// TwinCAT 3 PLC project NCInterpolation
// ProgramVersion: 3.1.0.8
// libraries:
//   Tc2_MC2, * (Beckhoff Automation GmbH)
//   Tc2_NCI, * (Beckhoff Automation GmbH)
//   Tc2_PlcInterpolation, * (Beckhoff Automation GmbH)
//   Tc2_Standard, * (Beckhoff Automation GmbH)
//   Tc2_System, * (Beckhoff Automation GmbH)
//   Tc3_Module, * (Beckhoff Automation GmbH)
// project tree:
//   GVLs/ GVL.TcGVL
//   / PlcTask.TcTTO
//   POUs/ Interpolate.TcPOU, MAIN.TcPOU, P_UML_Grafcet_Sequence.TcPOU
// real-time tasks:
//   TASK PlcTask: cycle T#10ms, priority 20, ADS port 350
// motion (NC):
//   TASK NC-Task 1 SAF: cycle T#5ms, priority 4, ADS port 501
//   TASK NC-Task 1 SVB: cycle T#10ms, priority 9, ADS port 511
//   AXIS FaulHaber_X (id 2)
//     General: UnitName=°
//     Dynamic: Acceleration=1925.33, Deceleration=1925.33, Jerk=187.597, DelayTime=0.015
//     Velo: Maximum=38000
//     OtherSettings: AllowMotionCmdToSlave=true
//     encoder EncType=19
//       EncPara: ScaleFactorNumerator=360, ScaleFactorDenominator=3000, MaxCount=#xffffffff
//         Inc: RefSoftSyncMask=#x0000ffff
//     drive DrvType=16
//       DrvPara: MaxCount=#xffffffff
//         Analog: VeloReferenz=42000
//         TimeComp: TaskDelayCycles=1
//     controller CtrType=1
//       CtrPara: PriorControlFactor=1
//         PosDiffControl: Enable=false
//         Observer: BandWidth=20
//   AXIS Stepper (id 4)
//     General: UnitName=°
//     Dynamic: Acceleration=4600, Deceleration=4600, Jerk=21160, DelayTime=0.015
//     Velo: Maximum=3600
//     OtherSettings: AllowMotionCmdToSlave=true
//     encoder EncType=1
//       EncPara: ScaleFactorNumerator=360, ScaleFactorDenominator=12800
//         Inc: RefSoftSyncMask=#x0000ffff
//     drive DrvType=5
//       Analog: VeloReferenz=3600
//       TimeComp: TaskDelayCycles=1
//     controller CtrType=1
//       CtrPara: PriorControlFactor=1
//         PosDiffControl: Enable=false
//         Observer: BandWidth=20
//   AXIS Servo (id 5)
//     General: UnitName=°
//     Dynamic: Acceleration=17000, Deceleration=17000, Jerk=289000, DelayTime=0.015
//     Velo: Maximum=16000
//     OtherSettings: AllowMotionCmdToSlave=true
//     encoder EncType=1
//       EncPara: ScaleFactorNumerator=360, ScaleFactorDenominator=1048576
//     drive DrvType=5
//       Analog: VeloReferenz=18000
//       TimeComp: TaskDelayCycles=1
//     controller CtrType=1
//       CtrPara: PriorControlFactor=1
//         Observer: BandWidth=20
// I/O:
//   DEVICE Device 2 (EtherCAT) (disabled), AmsNetId 192.168.1.109.3.1
//     Term 24 (EK1100) [EK1100 EtherCAT Coupler (2A E-Bus)]
//       Term 27 (EL7201) [EL7201 1Ch. MDP742 Servo motor output stage (50V, 4A)]
//       Term 28 (EL7031) [EL7031 1Ch. Stepper motor output stage (24V, 1.5A)]
//       Term 28 (EL6601) [EL6601 1 Port Switch (Ethernet, CoE)]
//       Term 29 (EL6751) [EL6751 CANopen Master]
//       Term 30 (EL9011) [EL9011 End Terminal]
//   DEVICE Device 1 (EL6751) (disabled), AmsNetId 192.168.1.109.2.1
//     Box 26 (CANopen Slave)
// variable links:
//   NC-Task 1 SAF/Axes/FaulHaber_X <-> Device 1 (EL6751)/Box 26 (CANopen Slave)
//     Drive/Inputs/In/nState1 <-> TxPDO 1/Inputs/Statusword
//     Drive/Inputs/In/nState2 <-> TxPDO 1/Inputs/Statusword @bit 8
//     Drive/Outputs/Out/nCtrl1 <-> RxPDO 1/Outputs/Controlword
//     Drive/Outputs/Out/nCtrl2 <-> RxPDO 1/Outputs/Controlword @bit 8
//     Drive/Outputs/Out/nDataOut1 <-> RxPDO 1/Outputs/Target Position
//     Enc/Inputs/In/nDataIn1 <-> TxPDO 1/Inputs/Actual Position
//   NCInterpolation/NCInterpolation Instance <-> Device 1 (EL6751)/Box 26 (CANopen Slave)
//     PlcTask Inputs/GVL.CURRENT_ACTUAL <-> TxPDO 2/Inputs/Current Actual Limit
//     PlcTask Inputs/GVL.CURRENT_LIMIT <-> TxPDO 2/Inputs/Actual Current Limit
//     PlcTask Outputs/GVL.CCL <-> RxPDO 2/Outputs/CCL
//     PlcTask Outputs/GVL.PCL <-> RxPDO 2/Outputs/PCL
//   NCInterpolation/NCInterpolation Instance <-> NC-Task 1 SAF/Axes/FaulHaber_X
//     PlcTask Inputs/GVL.SERVO_AXIS[1].NcToPlc <-> Outputs/ToPlc
//     PlcTask Outputs/GVL.SERVO_AXIS[1].PlcToNc <-> Inputs/FromPlc
//   NCInterpolation/NCInterpolation Instance <-> NC-Task 1 SAF/Axes/Servo
//     PlcTask Inputs/GVL.SERVO_AXIS[3].NcToPlc <-> Outputs/ToPlc
//     PlcTask Outputs/GVL.SERVO_AXIS[3].PlcToNc <-> Inputs/FromPlc
//   NCInterpolation/NCInterpolation Instance <-> NC-Task 1 SAF/Axes/Stepper
//     PlcTask Inputs/GVL.SERVO_AXIS[2].NcToPlc <-> Outputs/ToPlc
//     PlcTask Outputs/GVL.SERVO_AXIS[2].PlcToNc <-> Inputs/FromPlc
//   NCInterpolation/NCInterpolation Instance <-> NC-Task 1 SAF/NCI 2
//     PlcTask Inputs/GVL.nciGRPin[1] <-> Outputs/ToPlc
//     PlcTask Outputs/GVL.nciGRPout[1] <-> Inputs/FromPlc

CONFIGURATION NCInterpolation
    RESOURCE PLC ON TwinCAT3
        TASK PlcTask(INTERVAL := T#10ms, PRIORITY := 20);
        PROGRAM MAIN WITH PlcTask : MAIN;
    END_RESOURCE
END_CONFIGURATION

// ---- GVLs/GVL.TcGVL
VAR_GLOBAL
	SERVO_AXIS 				: 	ARRAY[1..MAX_AXES] OF AXIS_REF;
	nciGRPout	AT %Q* 		: 	ARRAY[1..MAX_NciGroups] OF PLCTONC_NCICHANNEL_REF;
	nciGRPin	AT %I* 		: 	ARRAY[1..MAX_NciGroups] OF NCTOPLC_NCICHANNEL_REF;
	CURRENT_LIMIT 	AT %I* 	: 	UINT;
	CURRENT_ACTUAL 	AT %I* 	: 	UINT;
END_VAR
VAR_GLOBAL CONSTANT
	MAX_Axes 				: 	INT := 3;
	MAX_NciGroups			: 	INT := 1;
END_VAR
VAR_GLOBAL PERSISTENT
	PCL AT %Q* 				: 	UINT := 1400;
	CCL AT %Q* 				: 	UINT := 600;
END_VAR

// ---- POUs/MAIN.TcPOU
PROGRAM MAIN
VAR
	fbPower			: ARRAY[1..MAX_AXES] OF MC_Power;
	SEQUENCE		: INT := 0;
	bStart			: BOOL := FALSE;
	i				: INT;
	fbInterpolate 	: Interpolate;
	TO_X, TO_Y, TO_T,TO_VELOCITY : LREAL;
END_VAR

CASE SEQUENCE OF 
0:
	IF bStart THEN 
		SEQUENCE := 10;
		i := 1;
	END_IF
10:
	fbPower[i](
	Axis:= SERVO_AXIS[i], 
	Enable:= TRUE, 
	Enable_Positive:= TRUE, 
	Enable_Negative:= TRUE, 
	Override:= 100 );
	IF fbPower[i].Status THEN
		SEQUENCE := SEQUENCE + 1;
	END_IF
11:
	i := i + 1;
	IF i > MAX_AXES THEN 
		i := 0;
		SEQUENCE := SEQUENCE + 9;
		bStart := FALSE;
	ELSE
		SEQUENCE := SEQUENCE - 1;		
	END_IF
20:
	IF bStart THEN
		SEQUENCE := SEQUENCE + 10;
	END_IF
30:
	IF fbInterpolate.GoTo(1,1,2,3,TO_X,TO_Y,TO_T,TO_VELOCITY) = 100 THEN
		SEQUENCE := 20;
		bStart := FALSE;
	ELSE
		bStart := TRUE;
	END_IF
END_CASE


P_UML_Grafcet_Sequence();

END_PROGRAM

// ---- POUs/Interpolate.TcPOU
FUNCTION_BLOCK Interpolate
VAR_INPUT
END_VAR
VAR_OUTPUT
END_VAR
VAR
	nciGrpConfig 			: ARRAY[1..MAX_NciGroups] OF CfgBuildExt3DGroup;
	nciRemoveConfig			: ARRAY[1..MAX_NciGroups] OF CfgReconfigGroup;
	fbCreate_Table 			: ARRAY[1..MAX_NciGroups] OF FB_NciFeedTablePreparation;
	nciFeedTable 			: ARRAY[1..MAX_NciGroups] OF FB_NCIFEEDTABLE;
	//Table data
	nciTable 				: ARRAY[1..MAX_NciGroups] OF ST_NCIFEEDGROUPTABLE;
	stGeoStart				: ST_NciGeoStart;
	stGeoLine				: ARRAY[1..MAX_NciGroups] OF ST_NciGeoLine;
	stEndOfTables			: ST_NciEndOfTables;
		
	AXIS_X, AXIS_Y, AXIS_Z	: ARRAY[1..MAX_NciGroups] OF INT;
	internal_STATE			: ARRAY[1..MAX_NciGroups] OF INT := [MAX_NciGroups(0)];
END_VAR

;

METHOD PUBLIC GoTo : INT
VAR_INPUT
	GROUP								: UDINT;
	X, Y, Z 							: INT;
	POSITION_X, POSITION_Y, POSITION_Z 	: LREAL;
	VELOCITY 							: LREAL;
END_VAR
CASE internal_State[GROUP] OF
0:
	AXIS_X[GROUP] 	:= X;
	AXIS_Y[GROUP]  	:= Y;
	AXIS_Z[GROUP] 	:= Z;
	stGeoLine[GROUP] .fEndPosX	:= POSITION_X;
	stGeoLine[GROUP] .fEndPosY	:= POSITION_Y;
	stGeoLine[GROUP] .fEndPosZ	:= POSITION_Z;
	stGeoLine[GROUP] .fVelo		:= VELOCITY;
	internal_State[GROUP]		:= internal_State[GROUP] + 10;
10:
	nciGrpConfig[GROUP](
	bExecute:= TRUE, 
	nGroupId:= nciGRPin[GROUP].GrpId, 
	nXAxisId:= SERVO_AXIS[AXIS_X[GROUP]].NcToPlc.AxisId, 
	nYAxisId:= SERVO_AXIS[AXIS_Y[GROUP]].NcToPlc.AxisId, 
	nZAxisId:= SERVO_AXIS[AXIS_Z[GROUP]].NcToPlc.AxisId );
	IF NOT nciGrpConfig[GROUP] .bBusy AND NOT nciGrpConfig[GROUP] .bErr THEN 
		nciGrpConfig[GROUP]( bExecute:= FALSE );
		ItpSetOverridePercent(fOverridePercent:= 100, sPlcToNci:= nciGRPout[GROUP]);
		internal_State[GROUP] := internal_State[GROUP] + 10;
	END_IF
20:
	stGeoStart.fPosX := SERVO_AXIS[X].NcToPlc.ActPos;
	stGeoStart.fPosY := SERVO_AXIS[Y].NcToPlc.ActPos;
	stGeoStart.fPosZ := SERVO_AXIS[Z].NcToPlc.ActPos;
	fbCreate_Table[GROUP] (
	nEntryType		:= E_NciEntryTypeGeoStart, 
	pEntry			:= ADR(stGeoStart), 
	bResetTable		:= 	FALSE, 
	bResetAll		:= 	FALSE, 
	stFeedGroupTable:= nciTable[GROUP] );
	internal_State[GROUP] := internal_State[GROUP] + 1;
21:
	fbCreate_Table[GROUP] (
	nEntryType		:= E_NciEntryTypeGeoLine, 
	pEntry			:= ADR(stGeoLine[GROUP]), 
	bResetTable		:= 	FALSE, 
	bResetAll		:= 	FALSE, 
	stFeedGroupTable:= nciTable[GROUP] );
	internal_State[GROUP] := internal_State[GROUP] + 1;
22:
	fbCreate_Table[GROUP](
	nEntryType		:= E_NciEntryTypeEndOfTables, 
	pEntry			:= ADR(stEndOfTables), 
	bResetTable		:= 	FALSE, 
	bResetAll		:= 	FALSE, 
	stFeedGroupTable:= nciTable[GROUP] );
	internal_State[GROUP] := internal_State[GROUP] + 8;
30:
	nciFeedTable[GROUP](
		bExecute:= TRUE,
		bLogFeederEntries:= FALSE, 
		stFeedGroupTable:= nciTable[GROUP], 
		stNciToPlc:= nciGRPin[GROUP] );
	IF 	nciFeedTable[GROUP].bChannelDone THEN 
		nciFeedTable[GROUP](
			bExecute		:= FALSE,
			stFeedGroupTable:= nciTable[GROUP], 
			stNciToPlc		:= nciGRPin[GROUP] );
		fbCreate_Table[GROUP](  
			bResetAll		:= TRUE, 
			stFeedGroupTable:= nciTable[GROUP] );
		internal_State[GROUP] := internal_State[GROUP] + 10;
	END_IF
40:
	nciRemoveConfig[GROUP](
		bExecute:= TRUE, 
		nGroupId:= nciGRPin[GROUP].GrpId, 
		tTimeOut:= T#500MS );
	IF NOT nciRemoveConfig[GROUP].bBusy THEN
		nciRemoveConfig[GROUP](
			bExecute:= FALSE, 
			nGroupId:= nciGRPin[GROUP].GrpId, 
			tTimeOut:= T#500MS );
		internal_State[GROUP] := 0;
		GoTo := 100;
	END_IF
END_CASE
END_METHOD

END_FUNCTION_BLOCK

// ---- POUs/P_UML_Grafcet_Sequence.TcPOU
PROGRAM P_UML_Grafcet_Sequence
VAR
END_VAR

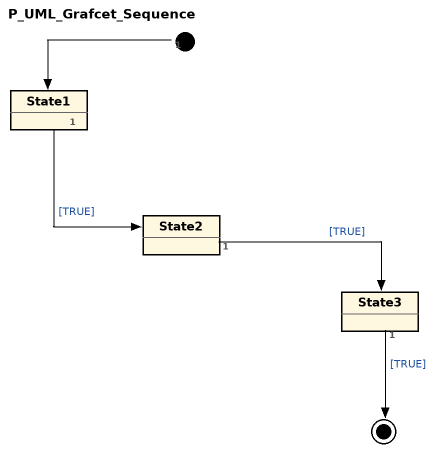
STATECHART P_UML_Grafcet_Sequence  // abortable
    START StartState1
    STATE State1
    STATE State2
    STATE State3
    END EndState1
    StartState1 -> State1  // priority 1, on completion
    State1 -> State2 [TRUE] // priority 1
    State2 -> State3 [TRUE] // priority 1
    State3 -> EndState1 [TRUE] // priority 1
END_STATECHART

END_PROGRAM
